// TIA Portal V15.1 export
// export: Created 2020-06-12T07:35:43.1943359Z, ExportSetting None, DisplayName Totally Integrated Automation Portal, DisplayVersion V15.1, DisplayName TIA Portal Openness, DisplayVersion V15.1, DisplayName STEP 7 Professional, DisplayVersion V15.1, DisplayName STEP 7 Safety, DisplayVersion V15.1, DisplayName WinCC Advanced, DisplayVersion V15.1
FUNCTION "CW_Pumps" : Void   // FC115, FBD
TITLE = CW Pumps handle
{ S7_Optimized_Access := 'TRUE' }
// stored: SetENOAutomatically False
   VAR_TEMP
      tBool : Bool;
      tOnM1 : Bool;
      tOnM2 : Bool;
      tOnM3 : Bool;
      tReqOn : Bool;
      tReqOff : Bool;
      tEmp_is_on : Bool;
      tPumpGLock : Bool;
      tPumpsReady : Bool;
      tPumpsArePrepared : Bool;
      tPumpsAreReleased : Bool;
      tPumpsTrip : Bool;
      tEconomOff : Bool;
      tPressOk : Bool;
      tPumpsLockStatus : Word;
      tPumpsSCond : Word;
      tPumpsCCond : Word;
      tPumpSpeedR : Real;
      tPumpSpeedMin : Real;
      tPumpSpeedMax : Real;
      tStage : Byte;
   END_VAR
   VAR_TEMP   // added for the SCL form of the ladder/FBD networks
      _w1 : Bool;
   END_VAR
BEGIN

REGION Network 1: TODO
END_REGION

REGION Network 2: HMI request treat
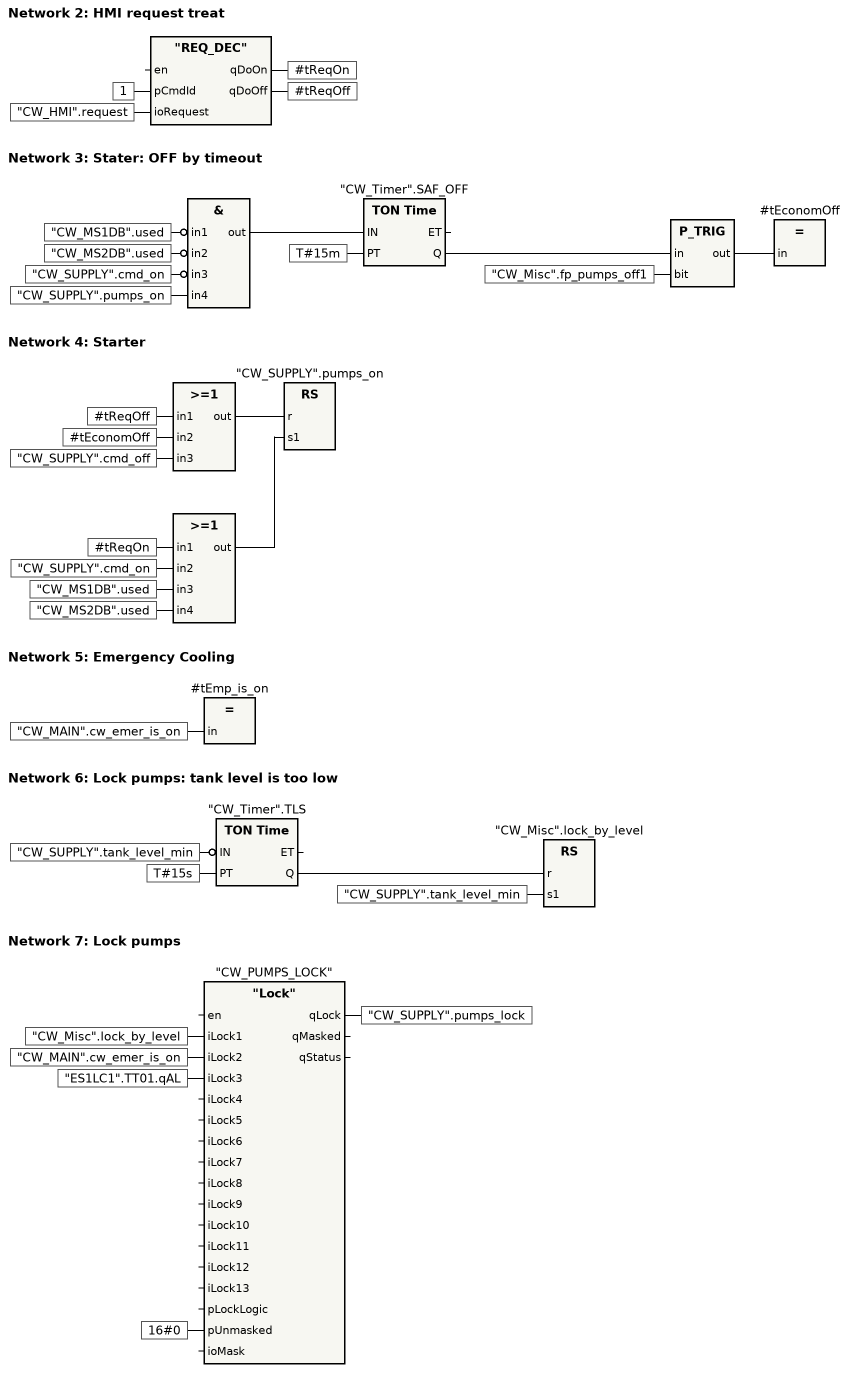
   "REQ_DEC"(pCmdId := 1, ioRequest := "CW_HMI".request, qDoOn => #tReqOn, qDoOff => #tReqOff);
END_REGION

REGION Network 3: Stater: OFF by timeout
   // Pum/Q: Why 2h delay?
   "CW_Timer".SAF_OFF.TON(IN := NOT "CW_MS1DB".used AND NOT "CW_MS2DB".used AND NOT "CW_SUPPLY".cmd_on AND "CW_SUPPLY".pumps_on,
                          PT := T#15m);
   #_w1 := "CW_Timer".SAF_OFF.Q AND NOT "CW_Misc".fp_pumps_off1;   // rising edge
   "CW_Misc".fp_pumps_off1 := "CW_Timer".SAF_OFF.Q;
   #tEconomOff := #_w1;
END_REGION

REGION Network 4: Starter
   IF #tReqOff OR #tEconomOff OR "CW_SUPPLY".cmd_off THEN
       "CW_SUPPLY".pumps_on := FALSE;   // RS flip-flop
   END_IF;
   IF #tReqOn OR "CW_SUPPLY".cmd_on OR "CW_MS1DB".used OR "CW_MS2DB".used THEN
       "CW_SUPPLY".pumps_on := TRUE;
   END_IF;
END_REGION

REGION Network 5: Emergency Cooling
   // Emergency power:
   // - diesel ()
   // - no one pump is running when neccessary
   #tEmp_is_on := "CW_MAIN".cw_emer_is_on;
END_REGION

REGION Network 6: Lock pumps: tank level is too low
   "CW_Timer".TLS.TON(IN := NOT "CW_SUPPLY".tank_level_min, PT := T#15s);
   IF "CW_Timer".TLS.Q THEN
       "CW_Misc".lock_by_level := FALSE;   // RS flip-flop
   END_IF;
   IF "CW_SUPPLY".tank_level_min THEN "CW_Misc".lock_by_level := TRUE; END_IF;
END_REGION

REGION Network 7: Lock pumps
   "CW_PUMPS_LOCK"(iLock1 := "CW_Misc".lock_by_level,   // "Lock"
                   iLock2 := "CW_MAIN".cw_emer_is_on,
                   iLock3 := "ES1LC1".TT01.qAL,
                   pUnmasked := 16#0,
                   qLock => "CW_SUPPLY".pumps_lock);
END_REGION

REGION Network 8: PUMPs: redundancy
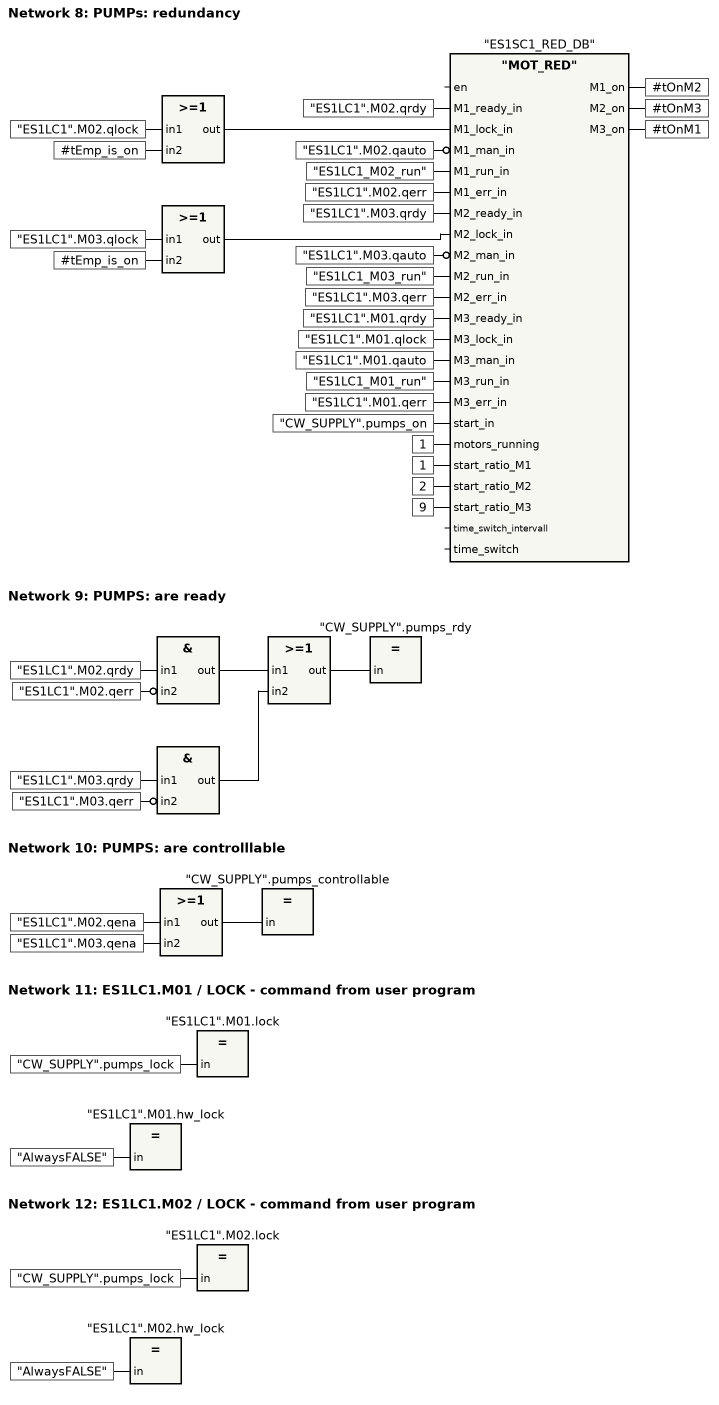
   "ES1SC1_RED_DB"(M1_ready_in := "ES1LC1".M02.qrdy,   // "MOT_RED"
                   M1_lock_in := "ES1LC1".M02.qlock OR #tEmp_is_on,
                   M1_man_in := NOT "ES1LC1".M02.qauto,
                   M1_run_in := "ES1LC1_M02_run",
                   M1_err_in := "ES1LC1".M02.qerr,
                   M2_ready_in := "ES1LC1".M03.qrdy,
                   M2_lock_in := "ES1LC1".M03.qlock OR #tEmp_is_on,
                   M2_man_in := NOT "ES1LC1".M03.qauto,
                   M2_run_in := "ES1LC1_M03_run",
                   M2_err_in := "ES1LC1".M03.qerr,
                   M3_ready_in := "ES1LC1".M01.qrdy,
                   M3_lock_in := "ES1LC1".M01.qlock,
                   M3_man_in := "ES1LC1".M01.qauto,
                   M3_run_in := "ES1LC1_M01_run",
                   M3_err_in := "ES1LC1".M01.qerr,
                   start_in := "CW_SUPPLY".pumps_on,
                   motors_running := 1,
                   start_ratio_M1 := 1,
                   start_ratio_M2 := 2,
                   start_ratio_M3 := 9,
                   M1_on => #tOnM2,
                   M2_on => #tOnM3,
                   M3_on => #tOnM1);
END_REGION

REGION Network 9: PUMPS: are ready
   "CW_SUPPLY".pumps_rdy := ("ES1LC1".M02.qrdy AND NOT "ES1LC1".M02.qerr) OR ("ES1LC1".M03.qrdy AND NOT "ES1LC1".M03.qerr);
END_REGION

REGION Network 10: PUMPS: are controlllable
   "CW_SUPPLY".pumps_controllable := "ES1LC1".M02.qena OR "ES1LC1".M03.qena;
END_REGION

REGION Network 11: ES1LC1.M01 / LOCK - command from user program
   "ES1LC1".M01.lock := "CW_SUPPLY".pumps_lock;
   "ES1LC1".M01.hw_lock := "AlwaysFALSE";
END_REGION

REGION Network 12: ES1LC1.M02 / LOCK - command from user program
   "ES1LC1".M02.lock := "CW_SUPPLY".pumps_lock;
   "ES1LC1".M02.hw_lock := "AlwaysFALSE";
END_REGION

REGION Network 13: ES1LC1.M03 / LOCK - command from user program
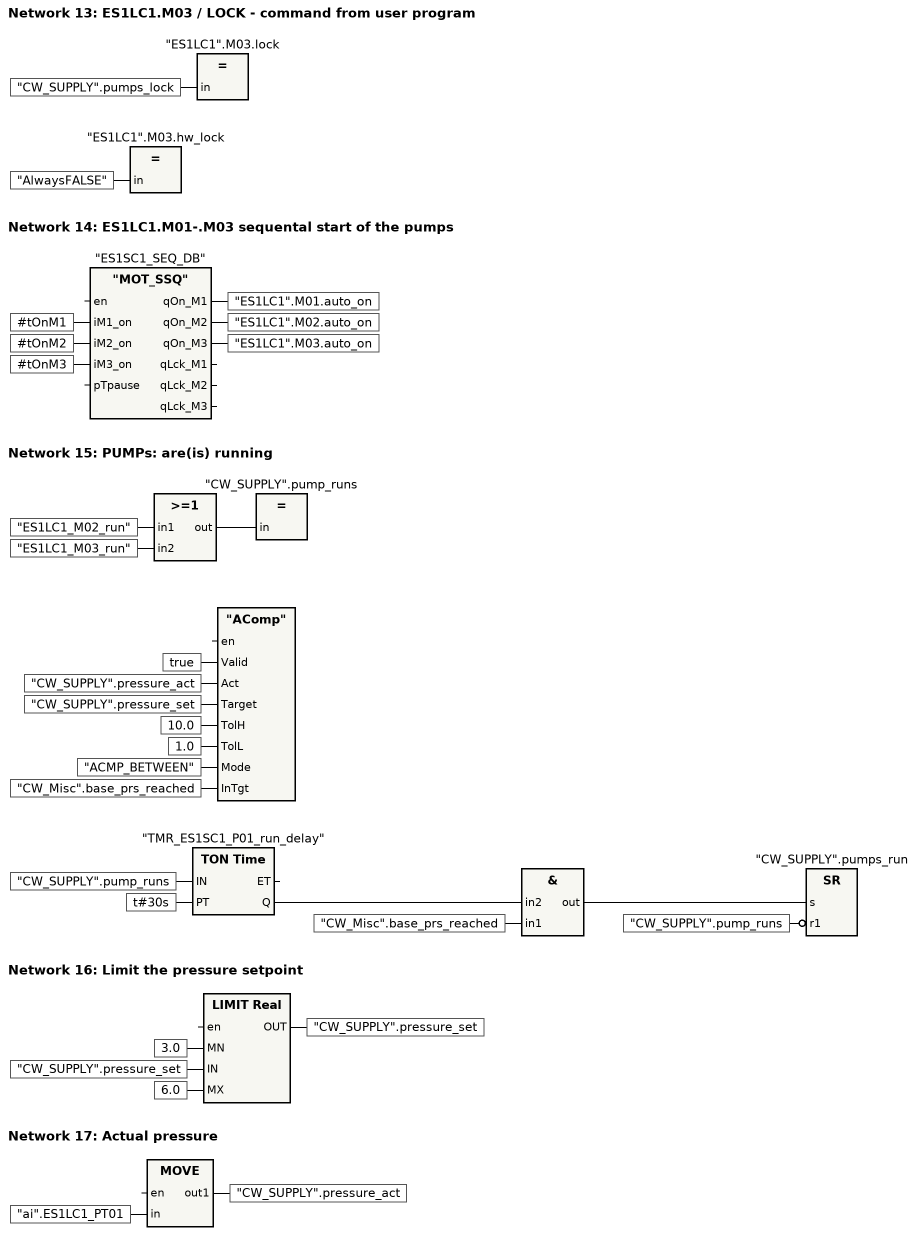
   "ES1LC1".M03.lock := "CW_SUPPLY".pumps_lock;
   "ES1LC1".M03.hw_lock := "AlwaysFALSE";
END_REGION

REGION Network 14: ES1LC1.M01-.M03 sequental start of the pumps
   "ES1SC1_SEQ_DB"(iM1_on := #tOnM1,   // "MOT_SSQ"
                   iM2_on := #tOnM2,
                   iM3_on := #tOnM3,
                   qOn_M1 => "ES1LC1".M01.auto_on,
                   qOn_M2 => "ES1LC1".M02.auto_on,
                   qOn_M3 => "ES1LC1".M03.auto_on);
END_REGION

REGION Network 15: PUMPs: are(is) running
   // The stable running state is delayed for a ramp time.
   // In this case the ramp time is 50s, we take 60s.
   "CW_SUPPLY".pump_runs := "ES1LC1_M02_run" OR "ES1LC1_M03_run";
   "AComp"(Valid := true,
           Act := "CW_SUPPLY".pressure_act,
           Target := "CW_SUPPLY".pressure_set,
           TolH := 10.0,
           TolL := 1.0,
           Mode := "ACMP_BETWEEN",
           InTgt := "CW_Misc".base_prs_reached);
   "TMR_ES1SC1_P01_run_delay".TON(IN := "CW_SUPPLY".pump_runs, PT := t#30s);
   IF "TMR_ES1SC1_P01_run_delay".Q AND "CW_Misc".base_prs_reached THEN
       "CW_SUPPLY".pumps_run := TRUE;   // SR flip-flop
   END_IF;
   IF NOT "CW_SUPPLY".pump_runs THEN "CW_SUPPLY".pumps_run := FALSE; END_IF;
END_REGION

REGION Network 16: Limit the pressure setpoint
   "CW_SUPPLY".pressure_set := LIMIT(MN := 3.0, IN := "CW_SUPPLY".pressure_set, MX := 6.0);
END_REGION

REGION Network 17: Actual pressure
   "CW_SUPPLY".pressure_act := "ai".ES1LC1_PT01;
END_REGION

REGION Network 18: Pressure control of pumps: PID
   // This block is only proxy. The real controller is in OB3x.
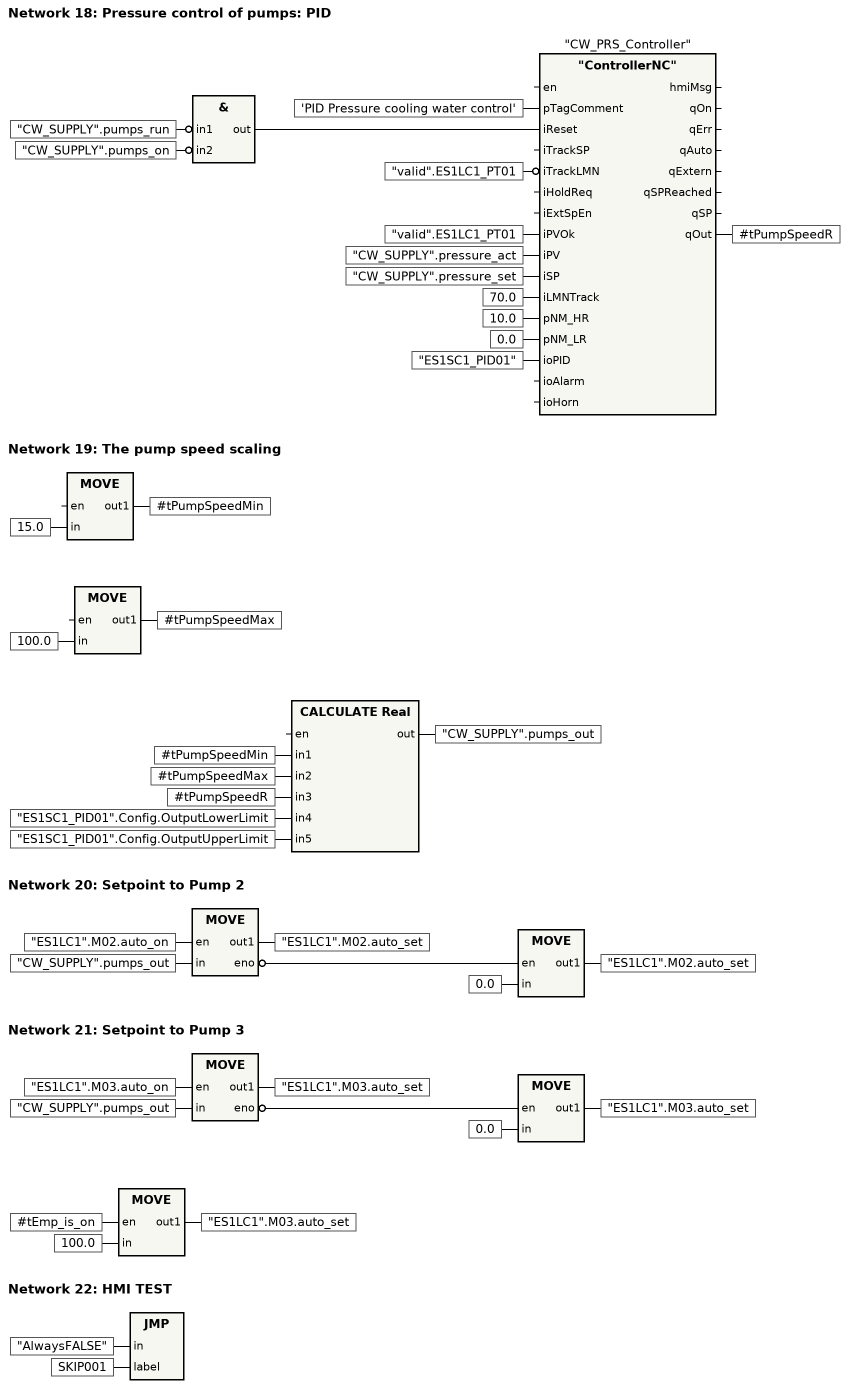
   "CW_PRS_Controller"(pTagComment := 'PID Pressure cooling water control',   // "ControllerNC"
                       iReset := NOT "CW_SUPPLY".pumps_run AND NOT "CW_SUPPLY".pumps_on,
                       iTrackLMN := NOT "valid".ES1LC1_PT01,
                       iPVOk := "valid".ES1LC1_PT01,
                       iPV := "CW_SUPPLY".pressure_act,
                       iSP := "CW_SUPPLY".pressure_set,
                       iLMNTrack := 70.0,
                       pNM_HR := 10.0,
                       pNM_LR := 0.0,
                       ioPID := "ES1SC1_PID01",
                       qOut => #tPumpSpeedR);
END_REGION

REGION Network 19: The pump speed scaling
   // We  need this because the pump cannot properly handle the speed lower then a some minimum
   #tPumpSpeedMin := 15.0;
   #tPumpSpeedMax := 100.0;
   "CW_SUPPLY".pumps_out := #tPumpSpeedMin + (#tPumpSpeedMax - #tPumpSpeedMin) * ((#tPumpSpeedR - "ES1SC1_PID01".Config.OutputLowerLimit) / ("ES1SC1_PID01".Config.OutputUpperLimit - "ES1SC1_PID01".Config.OutputLowerLimit));
END_REGION

REGION Network 20: Setpoint to Pump 2
   // ENO of a box is taken as its EN; it also drops when the box reports an error
   IF "ES1LC1".M02.auto_on THEN "ES1LC1".M02.auto_set := "CW_SUPPLY".pumps_out; END_IF;
   IF NOT "ES1LC1".M02.auto_on THEN "ES1LC1".M02.auto_set := 0.0; END_IF;
END_REGION

REGION Network 21: Setpoint to Pump 3
   // ENO of a box is taken as its EN; it also drops when the box reports an error
   IF "ES1LC1".M03.auto_on THEN "ES1LC1".M03.auto_set := "CW_SUPPLY".pumps_out; END_IF;
   IF NOT "ES1LC1".M03.auto_on THEN "ES1LC1".M03.auto_set := 0.0; END_IF;
   IF #tEmp_is_on THEN "ES1LC1".M03.auto_set := 100.0; END_IF;
END_REGION

REGION Network 22: HMI TEST
   // This network is used for HMI test
   IF "AlwaysFALSE" THEN GOTO SKIP001; END_IF;
END_REGION

REGION Network 23: HMI: STATUS
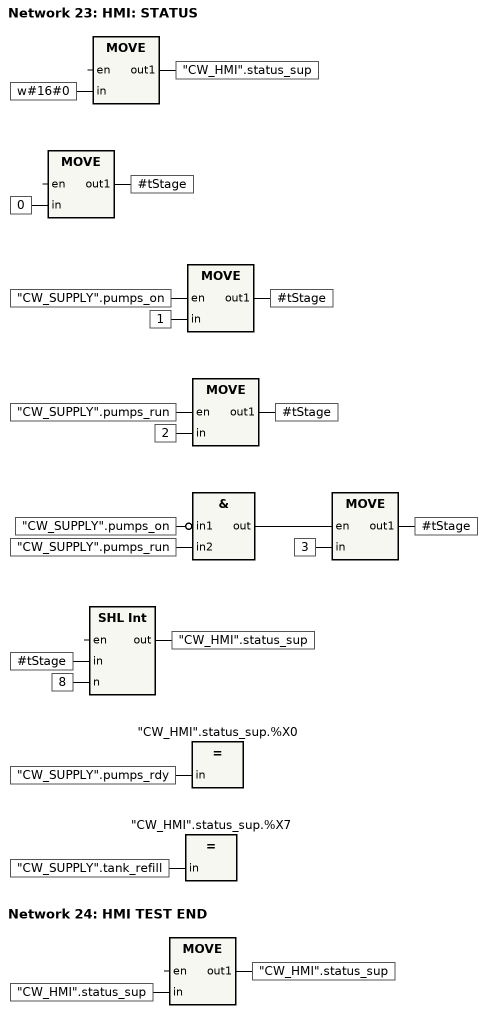
   "CW_HMI".status_sup := w#16#0;
   #tStage := 0;
   IF "CW_SUPPLY".pumps_on THEN #tStage := 1; END_IF;
   IF "CW_SUPPLY".pumps_run THEN #tStage := 2; END_IF;
   IF NOT "CW_SUPPLY".pumps_on AND "CW_SUPPLY".pumps_run THEN #tStage := 3; END_IF;
   "CW_HMI".status_sup := SHL(IN := #tStage, N := 8);
   "CW_HMI".status_sup.%X0 := "CW_SUPPLY".pumps_rdy;
   "CW_HMI".status_sup.%X7 := "CW_SUPPLY".tank_refill;
END_REGION

REGION Network 24: HMI TEST END
   SKIP001:
   "CW_HMI".status_sup := "CW_HMI".status_sup;
END_REGION

REGION Network 25: [[END]]
END_REGION
END_FUNCTION
